FUNCTION_BLOCK SRSection
  (* Standard: 61499-2 *)
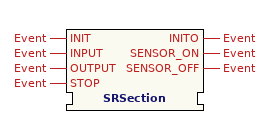
  EVENT_INPUT
    INIT;
    INPUT;
    OUTPUT;
    STOP;
  END_EVENT
  EVENT_OUTPUT
    INITO;
    SENSOR_ON;
    SENSOR_OFF;
  END_EVENT
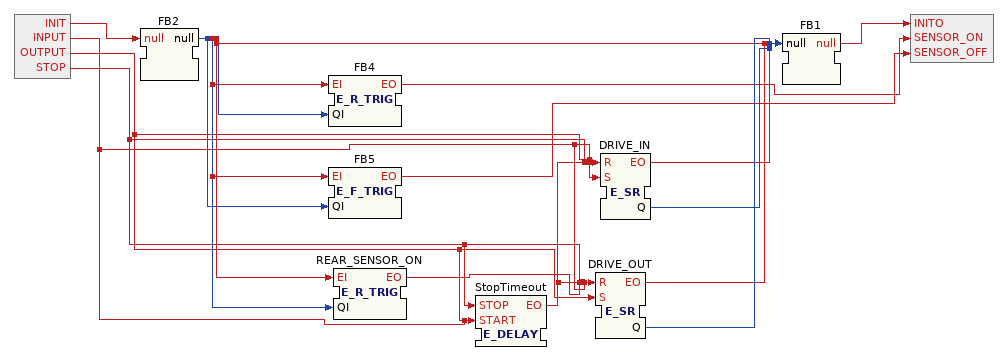
  FBS
    FB1 : ;
    FB2 : ;
    DRIVE_IN : E_SR;
    FB4 : E_R_TRIG;
    FB5 : E_F_TRIG;
    StopTimeout : E_DELAY;
    DRIVE_OUT : E_SR;
    REAR_SENSOR_ON : E_R_TRIG;
  END_FBS
  EVENT_CONNECTIONS
    FB4.EO TO SENSOR_ON;
    FB5.EO TO SENSOR_OFF;
    StopTimeout.EO TO DRIVE_IN.R;
    INIT TO FB2.null;
    FB2.null TO FB4.EI;
    FB2.null TO FB5.EI;
    FB2.null TO FB1.null;
    DRIVE_IN.EO TO FB1.null;
    FB1.null TO INITO;
    DRIVE_OUT.EO TO FB1.null;
    StopTimeout.EO TO DRIVE_OUT.R;
    INPUT TO DRIVE_IN.S;
    OUTPUT TO DRIVE_OUT.S;
    STOP TO DRIVE_IN.R;
    STOP TO StopTimeout.STOP;
    STOP TO DRIVE_OUT.R;
    OUTPUT TO DRIVE_IN.R;
    INPUT TO DRIVE_OUT.R;
    INPUT TO StopTimeout.START;
    OUTPUT TO StopTimeout.START;
    FB2.null TO REAR_SENSOR_ON.EI;
    REAR_SENSOR_ON.EO TO DRIVE_OUT.R;
  END_CONNECTIONS
  DATA_CONNECTIONS
    FB2.null TO FB4.QI;
    FB2.null TO FB5.QI;
    DRIVE_IN.Q TO FB1.null;
    DRIVE_OUT.Q TO FB1.null;
    FB2.null TO REAR_SENSOR_ON.QI;
  END_CONNECTIONS
END_FUNCTION_BLOCK
